SUBAPPLICATION Uebung_074_AX (* RPTO auf UT ausgeben (Adapter Version) mit Fendt-Schaltung *)
  (* Standard: 61499-2; Description: Copyright (c) 2023 Meisterschulen am Ostbahnhof This program and the accompanying materials are made available under the terms of the Eclipse Public License 2.0 which is available at https://www.eclipse.org/legal/epl-2.0/ SPDX-License-Identifier: EPL-2.0 *)
  (* Version 1.0, 2026-04-19, Franz Höpfinger, Meisterschulen am Ostbahnhof, initial API and implementation (Adapter Version of Uebung_074) *)
  PACKAGE Uebungen;
  IMPORT Uebungen::const::UT::TECU::DefaultPool_TECU::NumberVariable_Rear_PTO_output_shaft_speed;
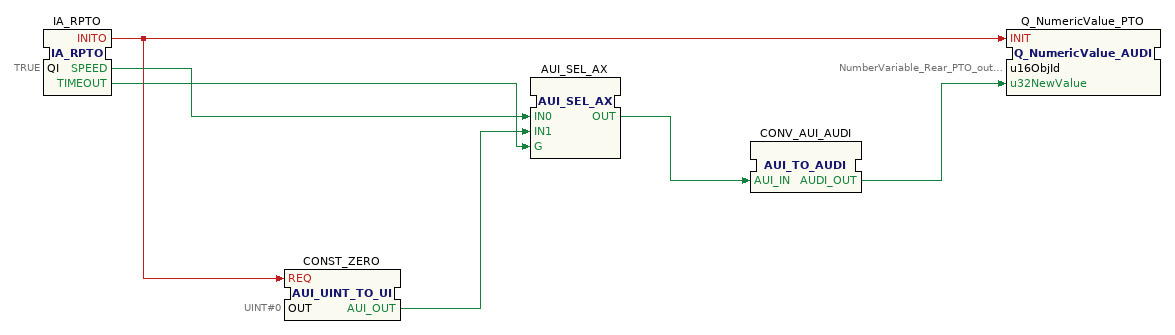
  (* "Fendt" Schaltung via Adapter: Bei Timeout wird 0 angezeigt! *)
  FBS
    IA_RPTO : isobus::tecu::IA_RPTO(QI := TRUE);
    Q_NumericValue_PTO : isobus::UT::Q::Q_NumericValue_AUDI(u16ObjId := NumberVariable_Rear_PTO_output_shaft_speed);
    AUI_SEL_AX : adapter::iec61131::selection::AUI_SEL_AX;
    CONST_ZERO : adapter::conversion::unidirectional::AUI_UINT_TO_UI(OUT := UINT#0);
    CONV_AUI_AUDI : adapter::conversion::unidirectional::AUI_TO_AUDI;
  END_FBS
  EVENT_CONNECTIONS
    IA_RPTO.INITO TO Q_NumericValue_PTO.INIT;
    IA_RPTO.INITO TO CONST_ZERO.REQ;
  END_CONNECTIONS
  ADAPTER_CONNECTIONS
    IA_RPTO.SPEED TO AUI_SEL_AX.IN0;
    CONST_ZERO.AUI_OUT TO AUI_SEL_AX.IN1;
    IA_RPTO.TIMEOUT TO AUI_SEL_AX.G;
    AUI_SEL_AX.OUT TO CONV_AUI_AUDI.AUI_IN;
    CONV_AUI_AUDI.AUDI_OUT TO Q_NumericValue_PTO.u32NewValue;
  END_CONNECTIONS
END_SUBAPPLICATION
